{attribute addProperty BoxType "EK1100-0000-0018"}
{attribute addProperty Id "Beckhoff_ER5xxxEK1122Beckhoff_ER5xxxEK1122_8A557ABF50262.75"}
{attribute addProperty CRC "454452707"}
{attribute addProperty SizeInBites "502"}
{attribute addProperty SizeInBytes "62.75"}
TYPE Beckhoff_ER5xxx_1B1665E3 EXTENDS EK1100_179A0949 :
STRUCT
	{attribute addProperty Name "Beckhoff_ER5xxxEK1122"}
	Beckhoff_ER5xxxEK1122 : Beckhoff_ER5xxxEK1122_8A557ABF;
END_STRUCT
END_TYPE

(* stored: Version 1.2.0.0, ProductVersion 3.1.4024.9
   DUT Beckhoff_ER5xxx_1B1665E3: Id {8e6945d4-7028-4f6f-9f9b-c74e686cd02a} *)
